FUNCTION_BLOCK FB_LoadCell IMPLEMENTS I_LoadCell
VAR
	//実I/Oと接続
	diBridgeInputs				:DINT;
	diSupplyInputs				:DINT;
	
	//演算後の入力値
	lrBridgeVoltage				:LREAL;
	lrSupplyVoltage				:LREAL;
	
	//測定重量と風袋重量
	lrGrossWeight				:LREAL;
	lrNetWeight					:LREAL;
	lrTareWeight				:REFERENCE TO LREAL;
	lrCalibrationWeight			:LREAL;	
	
	//ロードセルの仕様
	stLoadCellSpecification		:ST_LoadCellSpecification;
	
	//校正後の傾き
	lrSlope						:LREAL;
END_VAR

WeightMeasurement();

{warning 'メソッド実装を追加'}
METHOD CalibrationWeightSet
VAR
	lrNowGrossWeight				:LREAL;
END_VAR
	//今のグロスウェイト確認[kg]
	IF lrSupplyVoltage<>0 AND stLoadCellSpecification.lrRatedOutput<>0 THEN
		lrNowGrossWeight:=((DINT_TO_LREAL(diBridgeInputs)*20.0)/(DINT_TO_LREAL(diSupplyInputs)*12.0))*(stLoadCellSpecification.lrRatedCapacity/stLoadCellSpecification.lrRatedOutput);
	END_IF
	
	//今のグロスウェイトが風袋重量より重いことを確認
	IF lrTareWeight+0.010 < lrNowGrossWeight THEN
		//切片を計算
		IF lrNowGrossWeight<>0 AND lrTareWeight<>0 THEN
			lrSlope:=(lrCalibrationWeight-0)/(lrNowGrossWeight-lrTareWeight);
		END_IF
	END_IF
END_METHOD

{warning 'プロパティ実装を追加'}
PROPERTY diBridgeInputsProp : DINT
SET
diBridgeInputs:=diBridgeInputsProp;
END_SET
END_PROPERTY

{warning 'プロパティ実装を追加'}
PROPERTY diSupplyInputsProp : DINT
SET
diSupplyInputs:=diSupplyInputsProp;
END_SET
END_PROPERTY

{warning 'プロパティ実装を追加'}
PROPERTY lrBridgeVoltageProp : LREAL
GET
lrBridgeVoltageProp:=lrBridgeVoltage;
END_GET
END_PROPERTY

{warning 'プロパティ実装を追加'}
PROPERTY lrCalibrationWeightProp : LREAL
SET
lrCalibrationWeight:=lrCalibrationWeightProp;
END_SET
END_PROPERTY

{warning 'プロパティ実装を追加'}
PROPERTY lrGrossWeightProp : LREAL
GET
lrGrossWeightProp:=lrGrossWeight;
END_GET
END_PROPERTY

{warning 'プロパティ実装を追加'}
PROPERTY lrNetWeightProp : LREAL
GET
lrNetWeightProp:=lrNetWeight;
END_GET
END_PROPERTY

{warning 'プロパティ実装を追加'}
PROPERTY lrSupplyVoltageProp : LREAL
GET
lrSupplyVoltageProp:=lrSupplyVoltage;
END_GET
END_PROPERTY

{warning 'プロパティ実装を追加'}
PROPERTY lrTareWeightProp : REFERENCE TO LREAL
SET
VAR
	bCheck :BOOL;
END_VAR
IF __ISVALIDREF(lrTareWeightProp)=TRUE THEN
	bCheck:=TRUE;
END_IF

lrTareWeight REF=lrTareWeightProp;
END_SET
END_PROPERTY

{warning 'プロパティ実装を追加'}
PROPERTY stLoadCellSpecificationProp : ST_LoadCellSpecification
SET
stLoadCellSpecification:=stLoadCellSpecificationProp;
END_SET
END_PROPERTY

{warning 'メソッド実装を追加'}
METHOD TareWeightSet
	//風袋重量セット[kg]
	IF lrSupplyVoltage<>0 AND stLoadCellSpecification.lrRatedOutput<>0 THEN
		lrTareWeight:=((DINT_TO_LREAL(diBridgeInputs)*20.0)/(DINT_TO_LREAL(diSupplyInputs)*12.0))*(stLoadCellSpecification.lrRatedCapacity/stLoadCellSpecification.lrRatedOutput);
	END_IF
END_METHOD

{warning 'メソッド実装を追加'}
METHOD WeightMeasurement
	//ロードセルの出力電圧計算[mV]
	lrBridgeVoltage:=DINT_TO_LREAL(diBridgeInputs)*(20.0/2147483647);
	
	//ロードセルへの印加電圧計算[V]
	lrSupplyVoltage:=DINT_TO_LREAL(diSupplyInputs)*(12.0/2147483647);
	
	//グロスウェイト計算[kg]
	IF lrSupplyVoltage<>0 AND stLoadCellSpecification.lrRatedOutput<>0 THEN
		lrGrossWeight:=(lrBridgeVoltage/lrSupplyVoltage)*(stLoadCellSpecification.lrRatedCapacity/stLoadCellSpecification.lrRatedOutput);
	END_IF
	
	//ネットウェイト計算[kg]
	lrNetWeight:=lrGrossWeight-lrTareWeight;
END_METHOD

END_FUNCTION_BLOCK

(* stored: Version 1.1.0.1, ProductVersion 3.1.4024.12
   POU FB_LoadCell: Id {0956b8bf-68cc-43c5-8995-ef78b567874c}, SpecialFunc None
   Method CalibrationWeightSet: Id {93f54278-cb31-49f4-bfc1-0775b8414e9c}
   Property diBridgeInputsProp: Id {5eff2143-0b1c-497c-9e3c-1920cad2766f}
   Set Set: Id {91dc734f-9f57-4882-bca8-e62a29010e12}
   Property diSupplyInputsProp: Id {756219d0-0232-4b98-949a-708d0320154a}
   Set Set: Id {cd110deb-7528-4f6b-a889-4cd934eb29c8}
   Property lrBridgeVoltageProp: Id {d3f760e8-41da-4ddc-b41c-ac4cddbe73bd}
   Get Get: Id {f4149a2a-aba5-4856-bbf3-39ae86be694b}
   Property lrCalibrationWeightProp: Id {e55771da-6757-4d73-a527-38b789a79d63}
   Set Set: Id {48ec29ea-ef1c-4f49-8b4a-9485fd0250be}
   Property lrGrossWeightProp: Id {8f9a0b05-6d4e-44ea-a328-5a0f8141a8da}
   Get Get: Id {62896a2e-2fba-4042-b7df-6cfb3676fd28}
   Property lrNetWeightProp: Id {f9feebdb-7d80-40b0-9659-026331130eb9}
   Get Get: Id {9192aaba-682f-4b2a-9c04-a538d57d343f}
   Property lrSupplyVoltageProp: Id {f553a0ac-7513-4c81-bf0f-a359b42baf45}
   Get Get: Id {b69cf58d-f6f5-463b-add2-575323fe50ab}
   Property lrTareWeightProp: Id {db5e90bc-ae93-4279-baa9-42081ae45b8f}
   Set Set: Id {f22ff1e2-be44-4e4a-886a-e6c37f4f4282}
   Property stLoadCellSpecificationProp: Id {a84a2845-c8f0-4433-984d-1e6ece6dee2b}
   Set Set: Id {7ce3fc22-d897-4353-bd5d-f9e9ff3e4dfd}
   Method TareWeightSet: Id {0eed874b-e426-4c5c-96b2-9198e67a49d2}
   Method WeightMeasurement: Id {daeaec2b-19b4-41e3-b3a1-8d03e5dc53c7} *)
